// TwinCAT 3 PLC project M1L1_PLC
// ProgramVersion: 3.1.4020.5
// libraries:
//   Tc2_MC2, * (Beckhoff Automation GmbH)
//   Tc2_SerialCom, * (Beckhoff Automation GmbH)
//   Tc2_Standard, * (Beckhoff Automation GmbH)
//   Tc2_System, * (Beckhoff Automation GmbH)
//   Tc2_Utilities, * (Beckhoff Automation GmbH)
//   Tc3_Module, * (Beckhoff Automation GmbH)
//   VisuDialogs, * (System)
//   lcls-twincat-motion,0.0.0,SLAC
// project tree:
//   Common/POUs/Helpers/ FB_PI_E621_SerialDriver.TcPOU (not stored), FB_PI_E621_SerialTransaction.TcPOU (not stored)
//   DUTs/ DUT_MotionStage_Extras.TcDUT (not stored), ST_PiezoAxis.TcDUT (not stored)
//   / GlobalTextList.TcGTLO, PlcTask.TcTTO (not stored), serial_com.TcTTO, Visualization Manager.TcVMO (not stored)
//   GVLs/ GVL_SerialIO.TcGVL (not stored)
//   POUs/ MAIN.TcPOU
//   POUs/Serial Comm/ PiezoSerial.TcPOU, P_Serial_Com.TcPOU
//   VISUs/ Visualization.TcVIS, VISU_MotionStage.TcVIS (not stored)
// real-time tasks:
//   TASK PlcTask: cycle T#10ms, priority 20, ADS port 350
//   TASK serial_com: cycle T#10ms, priority 21, ADS port 351
// motion (NC):
//   TASK NC-Task 1 SAF: cycle T#2ms, priority 4, ADS port 501
//   TASK NC-Task 1 SVB: cycle T#10ms, priority 8, ADS port 511
//   AXIS y_up (id 6)
//     General: UnitName=um
//     Dynamic: Acceleration=5050, Deceleration=5050, Jerk=5100500, DelayTime=0.008
//     Velo: Maximum=100
//     OtherSettings: AllowMotionCmdToSlave=true
//     encoder EncType=29
//       EncPara: ScaleFactorNumerator=1, ScaleFactorDenominator=1000, MaxCount=#xffffffff, ReferenceSystem=1
//         SoftEndMinControl: Enable=true, Range=7200
//         SoftEndMaxControl: Enable=true, Range=100000
//         Inc: RefSoftSyncMask=#x0000ffff
//     drive DrvType=24
//       DrvPara: Inverse=true
//         Analog: VeloReferenz=500
//         TimeComp: TaskDelayCycles=1
//     controller CtrType=3
//       CtrPara: PriorControlFactor=1
//         PosDiffControl: Range=50, Time=0.2
//         PID: PosTn=0.005, PosIOutputLimit=0.0001, PosDOutputLimit=0, PosIDisableWhenMoving=true, DeadBandPosition=0.001
//         Observer: BandWidth=20
//   AXIS y_dwn (id 7)
//     General: UnitName=um
//     Dynamic: Acceleration=5050, Deceleration=5050, Jerk=5100500, DelayTime=0.008
//     Velo: Maximum=100
//     OtherSettings: AllowMotionCmdToSlave=true
//     encoder EncType=29
//       EncPara: ScaleFactorNumerator=1, ScaleFactorDenominator=1000, MaxCount=#xffffffff, ReferenceSystem=1
//         SoftEndMinControl: Enable=true, Range=10100
//         SoftEndMaxControl: Enable=true, Range=102600
//         Inc: RefSoftSyncMask=#x0000ffff
//     drive DrvType=24
//       DrvPara: Inverse=true
//         Analog: VeloReferenz=500
//         TimeComp: TaskDelayCycles=1
//     controller CtrType=3
//       CtrPara: PriorControlFactor=1
//         PosDiffControl: Range=50, Time=0.2
//         PID: PosTn=0.005, PosIOutputLimit=0.0001, PosDOutputLimit=0, PosIDisableWhenMoving=true, DeadBandPosition=0.001
//         Observer: BandWidth=20
//   AXIS x_up (id 1)
//     General: UnitName=um
//     Dynamic: Acceleration=1000, Deceleration=1000, DelayTime=0.008
//     Velo: Maximum=300
//     OtherSettings: AllowMotionCmdToSlave=true
//     encoder EncType=29
//       EncPara: ScaleFactorNumerator=0.001, MaxCount=#xffffffff, ReferenceSystem=1
//         SoftEndMinControl: Enable=true, Range=16900
//         SoftEndMaxControl: Enable=true, Range=23600
//         Inc: RefSoftSyncMask=#x0000ffff
//     drive DrvType=24
//       DrvPara: Inverse=true
//         Analog: VeloReferenz=625, ScaleFactorActTorque=0.1
//         TimeComp: TaskDelayCycles=1
//     controller CtrType=3
//       CtrPara: PriorControlFactor=1
//         PosDiffControl: Range=50
//         PID: PosTn=0.005, PosIOutputLimit=0.0001, PosDOutputLimit=0, PosIDisableWhenMoving=true, DeadBandPosition=0.001
//         Observer: BandWidth=20
//   AXIS x_dwn (id 9)
//     General: UnitName=um
//     Dynamic: AccelerationMaximum=1000, DecelerationMaximum=1000, Acceleration=1000, Deceleration=1000, Jerk=5000, DelayTime=0.008
//     Velo: Maximum=300
//     OtherSettings: AllowMotionCmdToSlave=true
//     encoder EncType=29
//       EncPara: ScaleFactorNumerator=0.001, MaxCount=#xffffffff
//         SoftEndMinControl: Enable=true, Range=15800
//         SoftEndMaxControl: Enable=true, Range=22600
//         Inc: RefSoftSyncMask=#x0000ffff
//     drive DrvType=24
//       Analog: VeloReferenz=625
//       TimeComp: TaskDelayCycles=1
//     controller CtrType=3
//       CtrPara: PriorControlFactor=1
//         PosDiffControl: Range=50, Time=0.2
//         PID: PosTn=0.005, PosIOutputLimit=0.0001, PosDOutputLimit=0, PosIDisableWhenMoving=true, DeadBandPosition=0.001
//         Observer: BandWidth=20
//   AXIS pitch (id 10)
//     General: UnitName=urad
//     Dynamic: Acceleration=64082.2, Deceleration=64082.2, Jerk=711156, DelayTime=0.008
//     Velo: Maximum=50
//     OtherSettings: AllowMotionCmdToSlave=true
//     encoder EncType=29
//       EncPara: ScaleFactorNumerator=0.00556, MaxCount=#xffffffff, ReferenceSystem=1
//         SoftEndMinControl: Enable=true, Range=57500
//         SoftEndMaxControl: Enable=true, Range=58900
//         ActPosCorrection: Time=0.008
//         Inc: RefSoftSyncMask=#x0000ffff
//     drive DrvType=24
//       DrvPara: Inverse=true
//         Analog: VeloReferenz=550
//         TimeComp: TaskDelayCycles=1
//     controller CtrType=3
//       CtrPara: PriorControlFactor=1
//         PosDiffControl: Range=15, Time=0.2
//         PID: PosKp=9, PosTn=0.0006, PosTv=1.2e-05, PosIOutputLimit=0.0005, PosDOutputLimit=0.0035, AccKa=0.001, DeadBandPosition=0.1
//         Observer: BandWidth=20
// I/O:
//   DEVICE Device 1 (EtherCAT)
//   DEVICE Device 4 (EtherCAT), AmsNetId 5.54.18.124.5.1
//     Term 4 (EK1100)
// variable links:
//   Axes/pitch <-> Device 4 (EtherCAT)/Term 4 (EK1100)/Term 10 (EL7047) - PitchCoarse
//     Drive/Inputs/In/nState1 @bit 3 <-> STM Status/Status/Error
//     Drive/Inputs/In/nState1 @bit 7 <-> STM Status/Status/Motor stall
//     Drive/Inputs/In/nState1 @bit 5 <-> STM Status/Status/Moving negative
//     Drive/Inputs/In/nState1 @bit 4 <-> STM Status/Status/Moving positive
//     Drive/Inputs/In/nState1 @bit 1 <-> STM Status/Status/Ready
//     Drive/Inputs/In/nState1 <-> STM Status/Status/Ready to enable
//     Drive/Inputs/In/nState1 @bit 6 <-> STM Status/Status/Torque reduced
//     Drive/Inputs/In/nState1 @bit 2 <-> STM Status/Status/Warning
//     Drive/Inputs/In/nState2 @bit 3 <-> STM Status/Status/Digital input 1
//     Drive/Inputs/In/nState2 @bit 4 <-> STM Status/Status/Digital input 2
//     Drive/Inputs/In/nState2 @bit 5 <-> STM Status/Status/Sync error
//     Drive/Inputs/In/nState2 @bit 7 <-> STM Status/Status/TxPDO Toggle
//     Drive/Inputs/In/nState4 @bit 1 <-> WcState/InputToggle
//     Drive/Inputs/In/nState4 <-> WcState/WcState
//     Drive/Outputs/Out/nCtrl1 <-> STM Control/Control/Enable
//     Drive/Outputs/Out/nCtrl1 @bit 2 <-> STM Control/Control/Reduce torque
//     Drive/Outputs/Out/nCtrl1 @bit 1 <-> STM Control/Control/Reset
//     Drive/Outputs/Out/nCtrl2 @bit 3 <-> STM Control/Control/Digital output 1
//     Drive/Outputs/Out/nDataOut2[0] <-> STM Velocity/Velocity
//   Axes/pitch <-> Device 4 (EtherCAT)/Term 4 (EK1100)/Term 13 (EL5042) - Pitch
//     Enc/Inputs/In/nComState @bit 1 <-> WcState/InputToggle
//     Enc/Inputs/In/nComState <-> WcState/WcState
//     Enc/Inputs/In/nDataIn1 <-> FB Inputs Channel 1/Position
//     Enc/Inputs/In/nState1 @bit 12 <-> FB Inputs Channel 1/Status/Diag
//     Enc/Inputs/In/nState1 @bit 1 <-> FB Inputs Channel 1/Status/Error
//     Enc/Inputs/In/nState1 @bit 14 <-> FB Inputs Channel 1/Status/Input cycle counter
//     Enc/Inputs/In/nState1 @bit 2 <-> FB Inputs Channel 1/Status/Ready
//     Enc/Inputs/In/nState1 @bit 13 <-> FB Inputs Channel 1/Status/TxPDO State
//     Enc/Inputs/In/nState1 <-> FB Inputs Channel 1/Status/Warning
//   Axes/x_dwn <-> Device 4 (EtherCAT)/Term 4 (EK1100)/Term 12 (EL5042) - X
//     Enc/Inputs/In/nComState @bit 1 <-> WcState/InputToggle
//     Enc/Inputs/In/nComState <-> WcState/WcState
//     Enc/Inputs/In/nDataIn1 <-> FB Inputs Channel 2/Position
//     Enc/Inputs/In/nState1 @bit 12 <-> FB Inputs Channel 2/Status/Diag
//     Enc/Inputs/In/nState1 @bit 1 <-> FB Inputs Channel 2/Status/Error
//     Enc/Inputs/In/nState1 @bit 14 <-> FB Inputs Channel 2/Status/Input cycle counter
//     Enc/Inputs/In/nState1 @bit 2 <-> FB Inputs Channel 2/Status/Ready
//     Enc/Inputs/In/nState1 @bit 13 <-> FB Inputs Channel 2/Status/TxPDO State
//     Enc/Inputs/In/nState1 <-> FB Inputs Channel 2/Status/Warning
//   Axes/x_dwn <-> Device 4 (EtherCAT)/Term 4 (EK1100)/Term 9 (EL7047) - Xdwn
//     Drive/Inputs/In/nState1 @bit 3 <-> STM Status/Status/Error
//     Drive/Inputs/In/nState1 @bit 7 <-> STM Status/Status/Motor stall
//     Drive/Inputs/In/nState1 @bit 5 <-> STM Status/Status/Moving negative
//     Drive/Inputs/In/nState1 @bit 4 <-> STM Status/Status/Moving positive
//     Drive/Inputs/In/nState1 @bit 1 <-> STM Status/Status/Ready
//     Drive/Inputs/In/nState1 <-> STM Status/Status/Ready to enable
//     Drive/Inputs/In/nState1 @bit 6 <-> STM Status/Status/Torque reduced
//     Drive/Inputs/In/nState1 @bit 2 <-> STM Status/Status/Warning
//     Drive/Inputs/In/nState2 @bit 3 <-> STM Status/Status/Digital input 1
//     Drive/Inputs/In/nState2 @bit 4 <-> STM Status/Status/Digital input 2
//     Drive/Inputs/In/nState2 @bit 5 <-> STM Status/Status/Sync error
//     Drive/Inputs/In/nState2 @bit 7 <-> STM Status/Status/TxPDO Toggle
//     Drive/Inputs/In/nState4 @bit 1 <-> WcState/InputToggle
//     Drive/Inputs/In/nState4 <-> WcState/WcState
//     Drive/Outputs/Out/nCtrl1 <-> STM Control/Control/Enable
//     Drive/Outputs/Out/nCtrl1 @bit 2 <-> STM Control/Control/Reduce torque
//     Drive/Outputs/Out/nCtrl1 @bit 1 <-> STM Control/Control/Reset
//     Drive/Outputs/Out/nCtrl2 @bit 3 <-> STM Control/Control/Digital output 1
//     Drive/Outputs/Out/nDataOut2[0] <-> STM Velocity/Velocity
//   Axes/y_dwn <-> Device 4 (EtherCAT)/Term 4 (EK1100)/Term 11 (EL5042) - Y
//     Enc/Inputs/In/nComState @bit 1 <-> WcState/InputToggle
//     Enc/Inputs/In/nComState <-> WcState/WcState
//     Enc/Inputs/In/nDataIn1 <-> FB Inputs Channel 2/Position
//     Enc/Inputs/In/nState1 @bit 12 <-> FB Inputs Channel 2/Status/Diag
//     Enc/Inputs/In/nState1 @bit 1 <-> FB Inputs Channel 2/Status/Error
//     Enc/Inputs/In/nState1 @bit 14 <-> FB Inputs Channel 2/Status/Input cycle counter
//     Enc/Inputs/In/nState1 @bit 2 <-> FB Inputs Channel 2/Status/Ready
//     Enc/Inputs/In/nState1 @bit 13 <-> FB Inputs Channel 2/Status/TxPDO State
//     Enc/Inputs/In/nState1 <-> FB Inputs Channel 2/Status/Warning
//   Axes/y_dwn <-> Device 4 (EtherCAT)/Term 4 (EK1100)/Term 7 (EL7047) - Ydwn
//     Drive/Inputs/In/nState1 @bit 3 <-> STM Status/Status/Error
//     Drive/Inputs/In/nState1 @bit 7 <-> STM Status/Status/Motor stall
//     Drive/Inputs/In/nState1 @bit 5 <-> STM Status/Status/Moving negative
//     Drive/Inputs/In/nState1 @bit 4 <-> STM Status/Status/Moving positive
//     Drive/Inputs/In/nState1 @bit 1 <-> STM Status/Status/Ready
//     Drive/Inputs/In/nState1 <-> STM Status/Status/Ready to enable
//     Drive/Inputs/In/nState1 @bit 6 <-> STM Status/Status/Torque reduced
//     Drive/Inputs/In/nState1 @bit 2 <-> STM Status/Status/Warning
//     Drive/Inputs/In/nState2 @bit 3 <-> STM Status/Status/Digital input 1
//     Drive/Inputs/In/nState2 @bit 4 <-> STM Status/Status/Digital input 2
//     Drive/Inputs/In/nState2 @bit 5 <-> STM Status/Status/Sync error
//     Drive/Inputs/In/nState2 @bit 7 <-> STM Status/Status/TxPDO Toggle
//     Drive/Inputs/In/nState4 @bit 1 <-> WcState/InputToggle
//     Drive/Inputs/In/nState4 <-> WcState/WcState
//     Drive/Outputs/Out/nCtrl1 <-> STM Control/Control/Enable
//     Drive/Outputs/Out/nCtrl1 @bit 2 <-> STM Control/Control/Reduce torque
//     Drive/Outputs/Out/nCtrl1 @bit 1 <-> STM Control/Control/Reset
//     Drive/Outputs/Out/nCtrl2 @bit 3 <-> STM Control/Control/Digital output 1
//     Drive/Outputs/Out/nDataOut2[0] <-> STM Velocity/Velocity
//   Axes/y_up <-> Device 4 (EtherCAT)/Term 4 (EK1100)/Term 11 (EL5042) - Y
//     Enc/Inputs/In/nComState @bit 1 <-> WcState/InputToggle
//     Enc/Inputs/In/nComState <-> WcState/WcState
//     Enc/Inputs/In/nDataIn1 <-> FB Inputs Channel 1/Position
//     Enc/Inputs/In/nState1 @bit 12 <-> FB Inputs Channel 1/Status/Diag
//     Enc/Inputs/In/nState1 @bit 1 <-> FB Inputs Channel 1/Status/Error
//     Enc/Inputs/In/nState1 @bit 14 <-> FB Inputs Channel 1/Status/Input cycle counter
//     Enc/Inputs/In/nState1 @bit 2 <-> FB Inputs Channel 1/Status/Ready
//     Enc/Inputs/In/nState1 @bit 13 <-> FB Inputs Channel 1/Status/TxPDO State
//     Enc/Inputs/In/nState1 <-> FB Inputs Channel 1/Status/Warning
//   Axes/y_up <-> Device 4 (EtherCAT)/Term 4 (EK1100)/Term 6 (EL7047) - Yup
//     Drive/Inputs/In/nState1 @bit 3 <-> STM Status/Status/Error
//     Drive/Inputs/In/nState1 @bit 7 <-> STM Status/Status/Motor stall
//     Drive/Inputs/In/nState1 @bit 5 <-> STM Status/Status/Moving negative
//     Drive/Inputs/In/nState1 @bit 4 <-> STM Status/Status/Moving positive
//     Drive/Inputs/In/nState1 @bit 1 <-> STM Status/Status/Ready
//     Drive/Inputs/In/nState1 <-> STM Status/Status/Ready to enable
//     Drive/Inputs/In/nState1 @bit 6 <-> STM Status/Status/Torque reduced
//     Drive/Inputs/In/nState1 @bit 2 <-> STM Status/Status/Warning
//     Drive/Inputs/In/nState2 @bit 3 <-> STM Status/Status/Digital input 1
//     Drive/Inputs/In/nState2 @bit 4 <-> STM Status/Status/Digital input 2
//     Drive/Inputs/In/nState2 @bit 5 <-> STM Status/Status/Sync error
//     Drive/Inputs/In/nState2 @bit 7 <-> STM Status/Status/TxPDO Toggle
//     Drive/Inputs/In/nState4 @bit 1 <-> WcState/InputToggle
//     Drive/Inputs/In/nState4 <-> WcState/WcState
//     Drive/Outputs/Out/nCtrl1 <-> STM Control/Control/Enable
//     Drive/Outputs/Out/nCtrl1 @bit 2 <-> STM Control/Control/Reduce torque
//     Drive/Outputs/Out/nCtrl1 @bit 1 <-> STM Control/Control/Reset
//     Drive/Outputs/Out/nCtrl2 @bit 3 <-> STM Control/Control/Digital output 1
//     Drive/Outputs/Out/nDataOut2[0] <-> STM Velocity/Velocity
//   (this object) <-> Device 4 (EtherCAT)/Term 4 (EK1100)/Term 12 (EL5042) - X
//     Enc/Inputs/In/nComState @bit 1 <-> WcState/InputToggle
//     Enc/Inputs/In/nComState <-> WcState/WcState
//     Enc/Inputs/In/nDataIn1 <-> FB Inputs Channel 1/Position
//     Enc/Inputs/In/nState1 @bit 12 <-> FB Inputs Channel 1/Status/Diag
//     Enc/Inputs/In/nState1 @bit 1 <-> FB Inputs Channel 1/Status/Error
//     Enc/Inputs/In/nState1 @bit 14 <-> FB Inputs Channel 1/Status/Input cycle counter
//     Enc/Inputs/In/nState1 @bit 2 <-> FB Inputs Channel 1/Status/Ready
//     Enc/Inputs/In/nState1 @bit 13 <-> FB Inputs Channel 1/Status/TxPDO State
//     Enc/Inputs/In/nState1 <-> FB Inputs Channel 1/Status/Warning
//   (this object) <-> Device 4 (EtherCAT)/Term 4 (EK1100)/Term 8 (EL7047) - Xup
//     Drive/Inputs/In/nState1 @bit 3 <-> STM Status/Error
//     Drive/Inputs/In/nState1 @bit 7 <-> STM Status/Motor stall
//     Drive/Inputs/In/nState1 @bit 5 <-> STM Status/Moving negative
//     Drive/Inputs/In/nState1 @bit 4 <-> STM Status/Moving positive
//     Drive/Inputs/In/nState1 @bit 1 <-> STM Status/Ready
//     Drive/Inputs/In/nState1 <-> STM Status/Ready to enable
//     Drive/Inputs/In/nState1 @bit 6 <-> STM Status/Torque reduced
//     Drive/Inputs/In/nState1 @bit 2 <-> STM Status/Warning
//     Drive/Inputs/In/nState2 @bit 3 <-> STM Status/Digital input 1
//     Drive/Inputs/In/nState2 @bit 4 <-> STM Status/Digital input 2
//     Drive/Inputs/In/nState2 @bit 5 <-> STM Status/Sync error
//     Drive/Inputs/In/nState2 @bit 7 <-> STM Status/TxPDO Toggle
//     Drive/Inputs/In/nState4 @bit 1 <-> WcState/InputToggle
//     Drive/Inputs/In/nState4 <-> WcState/WcState
//     Drive/Outputs/Out/nCtrl1 <-> STM Control/Enable
//     Drive/Outputs/Out/nCtrl1 @bit 2 <-> STM Control/Reduce torque
//     Drive/Outputs/Out/nCtrl1 @bit 1 <-> STM Control/Reset
//     Drive/Outputs/Out/nCtrl2 @bit 3 <-> STM Control/Digital output 1
//     Drive/Outputs/Out/nDataOut2[0] <-> STM Velocity/Velocity
//   M1L1_PLC Instance <-> Device 1 (EtherCAT)/Term 1 (EK1200)/Term 2 (EL1004)
//     PlcTask Inputs/MAIN.stoEnable1 <-> Channel 1/Input
//     PlcTask Inputs/MAIN.stoEnable2 <-> Channel 2/Input
//   M1L1_PLC Instance <-> Device 4 (EtherCAT)/Term 4 (EK1100)/Term 10 (EL7047) - PitchCoarse
//     PlcTask Inputs/MAIN.M5.bLimitBackwardEnable <-> STM Status/Status/Digital input 2
//     PlcTask Inputs/MAIN.M5.bLimitForwardEnable <-> STM Status/Status/Digital input 1
//   M1L1_PLC Instance <-> Device 4 (EtherCAT)/Term 4 (EK1100)/Term 11 (EL5042) - Y
//     PlcTask Inputs/MAIN.bEncWarningYdwn <-> FB Inputs Channel 2/Status/Warning
//     PlcTask Inputs/MAIN.bEncWarningYup <-> FB Inputs Channel 1/Status/Warning
//     PlcTask Inputs/MAIN.y_dwn_enc/Count <-> FB Inputs Channel 2/Position
//     PlcTask Inputs/MAIN.y_up_enc/Count <-> FB Inputs Channel 1/Position
//   M1L1_PLC Instance <-> Device 4 (EtherCAT)/Term 4 (EK1100)/Term 12 (EL5042) - X
//     PlcTask Inputs/MAIN.bEncWarningXdwn <-> FB Inputs Channel 2/Status/Warning
//     PlcTask Inputs/MAIN.x_dwn_enc/Count <-> FB Inputs Channel 2/Position
//     PlcTask Inputs/MAIN.x_up_enc/Count <-> FB Inputs Channel 1/Position
//   M1L1_PLC Instance <-> Device 4 (EtherCAT)/Term 4 (EK1100)/Term 13 (EL5042) - Pitch
//     PlcTask Inputs/MAIN.bEncWarningPitch <-> FB Inputs Channel 1/Status/Warning
//   M1L1_PLC Instance <-> Device 4 (EtherCAT)/Term 4 (EK1100)/Term 6 (EL7047) - Yup
//     PlcTask Inputs/MAIN.M1.bLimitBackwardEnable <-> STM Status/Status/Digital input 2
//     PlcTask Inputs/MAIN.M1.bLimitForwardEnable <-> STM Status/Status/Digital input 1
//   M1L1_PLC Instance <-> Device 4 (EtherCAT)/Term 4 (EK1100)/Term 7 (EL7047) - Ydwn
//     PlcTask Inputs/MAIN.M2.bLimitBackwardEnable <-> STM Status/Status/Digital input 2
//     PlcTask Inputs/MAIN.M2.bLimitForwardEnable <-> STM Status/Status/Digital input 1
//   M1L1_PLC Instance <-> Device 4 (EtherCAT)/Term 4 (EK1100)/Term 8 (EL7047) - Xup
//     PlcTask Inputs/MAIN.M3.bLimitBackwardEnable <-> STM Status/Digital input 2
//     PlcTask Inputs/MAIN.M3.bLimitForwardEnable <-> STM Status/Digital input 1
//   M1L1_PLC Instance <-> Device 4 (EtherCAT)/Term 4 (EK1100)/Term 9 (EL7047) - Xdwn
//     PlcTask Inputs/MAIN.M4.bLimitBackwardEnable <-> STM Status/Status/Digital input 2
//     PlcTask Inputs/MAIN.M4.bLimitForwardEnable <-> STM Status/Status/Digital input 1
//   M1L1_PLC Instance <-> NC-Task 1 SAF/Axes/pitch
//     PlcTask Inputs/MAIN.M5.Axis.NcToPlc <-> Outputs/ToPlc
//     PlcTask Outputs/MAIN.M5.Axis.PlcToNc <-> Inputs/FromPlc
//   M1L1_PLC Instance <-> NC-Task 1 SAF/Axes/x_dwn
//     PlcTask Inputs/MAIN.M4.Axis.NcToPlc <-> Outputs/ToPlc
//     PlcTask Outputs/MAIN.M4.Axis.PlcToNc <-> Inputs/FromPlc
//   M1L1_PLC Instance <-> NC-Task 1 SAF/Axes/x_up
//     PlcTask Inputs/MAIN.M3.Axis.NcToPlc <-> Outputs/ToPlc
//     PlcTask Outputs/MAIN.M3.Axis.PlcToNc <-> Inputs/FromPlc
//   M1L1_PLC Instance <-> NC-Task 1 SAF/Axes/y_dwn
//     PlcTask Inputs/MAIN.M2.Axis.NcToPlc <-> Outputs/ToPlc
//     PlcTask Outputs/MAIN.M2.Axis.PlcToNc <-> Inputs/FromPlc
//   M1L1_PLC Instance <-> NC-Task 1 SAF/Axes/y_up
//     PlcTask Inputs/MAIN.M1.Axis.NcToPlc <-> Outputs/ToPlc
//     PlcTask Outputs/MAIN.M1.Axis.PlcToNc <-> Inputs/FromPlc

CONFIGURATION M1L1_PLC
    RESOURCE PLC ON TwinCAT3
        TASK serial_com(INTERVAL := T#10ms, PRIORITY := 21);
        PROGRAM P_Serial_Com WITH serial_com : P_Serial_Com;
    END_RESOURCE
END_CONFIGURATION

// ---- POUs/Serial Comm/P_Serial_Com.TcPOU
PROGRAM P_Serial_Com
VAR
	fbSerialLineControl_EL6001_P1: SerialLineControl;
END_VAR

//These are the global IOs...don't forget to copy your data into them

(* EL6001 Serial port 0 com function *)
fbSerialLineControl_EL6001_P1(
	Mode:= SERIALLINEMODE_EL6_22B (*SERIALLINEMODE_KL6_22B_STANDARD*),
	pComIn:= ADR(Serial_P1_stComIn),
	pComOut:=ADR(Serial_P1_stComOut) ,
	SizeComIn:= SIZEOF(Serial_P1_stComIn),
	TxBuffer:= Serial_P1_SerialTXBuffer,
	RxBuffer:= Serial_P1_SerialRXBuffer,
	Error=> ,
	ErrorID=> );

END_PROGRAM

// ---- POUs/MAIN.TcPOU
PROGRAM MAIN
VAR
    M1: DUT_MotionStage:=(nCommand:=3); // Yup
	M2: DUT_MotionStage:=(nCommand:=3); // Ydwn
	M3: DUT_MotionStage:=(nCommand:=3); // Xup
	M4: DUT_MotionStage:=(nCommand:=3); // Xdwn
	M5: DUT_MotionStage:=(nCommand:=3); // PitchCoarse
	M1_Extras : DUT_MotionStage_Extras;
	M2_Extras : DUT_MotionStage_Extras;
	M3_Extras : DUT_MotionStage_Extras;
	M4_Extras : DUT_MotionStage_Extras;
	M5_Extras : DUT_MotionStage_Extras;

	fbMotionStage_x_up, fbMotionStage_x_dwn, fbMotionStage_y_up, fbMotionStage_y_dwn, fbMotionStage_pitch : FB_MotionStage;

	stoEnable1 AT %I* : BOOL;
	stoEnable2 AT %I* : BOOL;
	x_up_enc  AT %I*: ST_RenishawAbsEnc;
	x_dwn_enc  AT %I*: ST_RenishawAbsEnc;
	y_up_enc  AT %I*: ST_RenishawAbsEnc;
	y_dwn_enc  AT %I*: ST_RenishawAbsEnc;

	// Auto coupling function block
	fbAutoCoupleX : FB_GantryAutoCoupling;
	fbAutoCoupleY : FB_GantryAutoCoupling;
	bExecuteCoupleX : BOOL;
	bExecuteCoupleY : BOOL;
	bExecuteDecoupleX : BOOL;
	bExecuteDecoupleY : BOOL;
	bGantryAlreadyCoupledX : BOOL;
	bGantryAlreadyCoupledY : BOOL;
	
	// Gantry variables
	nCurrGantryX : LINT;
	nCurrGantryY : LINT;
	nGantryTolX : LINT := 75000;
	nGantryTolY : LINT := 75000;
	fCurrGantryX_um : LREAL;
	fCurrGantryY_um : LREAL;

	// Current Variables
	nCoilACurrRaw AT %I* : UINT;
	nCoilBCurrRaw AT %I* : UINT;
	nCoilACurr : INT;
	nCoilBCurr : INT;
	nTotCurr : INT;

	// Counters for encoder warning
	ctuXup : CTU;
	bEncWarningXup AT %I* : BOOL; // TRUE when encoder warning occurs
	nNumWarningsXup : WORD := 0;

	ctuXdwn : CTU;
	bEncWarningXdwn AT %I* : BOOL; // TRUE when encoder warning occurs
	nNumWarningsXdwn : WORD := 0;

	ctuYup : CTU;
	bEncWarningYup AT %I* : BOOL; // TRUE when encoder warning occurs
	nNumWarningsYup : WORD := 0;

	ctuYdwn : CTU;
	bEncWarningYdwn AT %I* : BOOL; // TRUE when encoder warning occurs
	nNumWarningsYdwn : WORD := 0;

	ctuPitch : CTU;
	bEncWarningPitch AT %I* : BOOL; // TRUE when encoder warning occurs
	nNumWarningsPitch : WORD := 0;
END_VAR

// M2K3
// Buttons to enable motors: write 0 to enable, 2 to disable
M1.nEnableMode; // Yup
M2.nEnableMode; // Ydwn
M3.nEnableMode; // Xup
M4.nEnableMode; // Xdwn
M5.nEnableMode; // PitchCoarse

// Encoder Reference Values: Initially took from Axilon FAT
// Had to realign encoders (lights were red) and so now using motor positions after aligning (lights turned blue)
// M2K3 Ref Vals
(*
y_up_enc.Ref := 43575680;
y_dwn_enc.Ref := 46974520;
x_up_enc.Ref := 20359920;
x_dwn_enc.Ref := 19780970;
*)
// Gantry zero positions after realignment with metrology
y_up_enc.Ref := 40653120;
y_dwn_enc.Ref := 43456180;
x_up_enc.Ref := 23635520;
x_dwn_enc.Ref := 22541650;

// Gantry Differences to monitor
nCurrGantryY := ((ULINT_TO_LINT(y_up_enc.Count) - ULINT_TO_LINT(y_up_enc.Ref)) - (ULINT_TO_LINT(y_dwn_enc.Count) - ULINT_TO_LINT(y_dwn_enc.Ref)));
nCurrGantryX := ((ULINT_TO_LINT(x_up_enc.Count) - ULINT_TO_LINT(x_up_enc.Ref)) - (ULINT_TO_LINT(x_dwn_enc.Count) - ULINT_TO_LINT(x_dwn_enc.Ref)));
fCurrGantryY_um := LINT_TO_LREAL(nCurrGantryY)/1000.0;
fCurrGantryx_um := LINT_TO_LREAL(nCurrGantryX)/1000.0;

// E-stop
M1.bHardwareEnable := stoEnable1 AND stoEnable2;
M2.bHardwareEnable := stoEnable1 AND stoEnable2;
M3.bHardwareEnable := stoEnable1 AND stoEnable2;
M4.bHardwareEnable := stoEnable1 AND stoEnable2;
M5.bHardwareEnable := stoEnable1 AND stoEnable2;


// Start Autocoupling
fbAutoCoupleX(nGantryTol:=nGantryTolX, Master:=M3, MasterEnc:=x_up_enc, Slave:=M4,
	          SlaveEnc:=x_dwn_enc, bExecuteCouple:=bExecuteCoupleX,
              bExecuteDecouple:=bExecuteDecoupleX,
              bGantryAlreadyCoupled=>bGantryAlreadyCoupledX);


fbAutoCoupleY(nGantryTol:=nGantryTolY, Master:=M1, MasterEnc:=y_up_enc, Slave:=M2,
	          SlaveEnc:=y_dwn_enc, bExecuteCouple:=bExecuteCoupleY,
              bExecuteDecouple:=bExecuteDecoupleY,
			  bGantryAlreadyCoupled=>bGantryAlreadyCoupledY);


fbMotionStage_y_up  (stMotionStage:=M1);
fbMotionStage_y_dwn (stMotionStage:=M2);
fbMotionStage_x_up  (stMotionStage:=M3);
fbMotionStage_x_dwn (stMotionStage:=M4);
fbMotionStage_pitch (stMotionStage:=M5);

// Record Coil Current
nCoilACurr := UINT_TO_INT(nCoilACurrRaw);
nCoilBCurr := UINT_TO_INT(nCoilBCurrRaw);
nTotCurr := ABS(nCoilACurr) + ABS(nCoilBCurr);

// Count when encoders throw warning
ctuXup(CU:=bEncWarningXup, CV=>nNumWarningsXup);
ctuXdwn(CU:=bEncWarningXdwn, CV=>nNumWarningsXdwn);
ctuYup(CU:=bEncWarningYup, CV=>nNumWarningsYup);
ctuYdwn(CU:=bEncWarningYdwn, CV=>nNumWarningsYdwn);
ctuPitch(CU:=bEncWarningPitch, CV=>nNumWarningsPitch);

END_PROGRAM

// ---- POUs/Serial Comm/PiezoSerial.TcPOU
PROGRAM PiezoSerial
VAR
	//PI Serial
	fbE621SerialDriverM1 : FB_PI_E621_SerialDriver;
	piezo: ST_PiezoAxis;
	rtInitParams	:	R_TRIG;
	tonTimeoutRstM1	: TON := (PT:=T#2S); //For timeout reset
	tonTimeoutRstM2	: TON := (PT:=T#2S); //For timeout reset
END_VAR

//M1 Piezo E-621
///////////////////////
	fbE621SerialDriverM1.i_xExecute := TRUE;
	fbE621SerialDriverM1.i_xExecute R= fbE621SerialDriverM1.q_xDone;
	fbE621SerialDriverM1(
		iq_stPiezoAxis:= piezo, 
		iq_stSerialRXBuffer:= Serial_P1_SerialRXBuffer, 
		iq_stSerialTXBuffer:= Serial_P1_SerialTXBuffer);

END_PROGRAM

// ---- GlobalTextList.TcGTLO
TEXTLIST GlobalTextList
  991 = '%f'
  359 = '%X'
  351 = '+'
  997 = '-'
  355 = '0 = Default Acceleration'
  357 = '0 = Default Deceleration'
  354 = 'Acceleration: %f'
  24 = 'Already Coupled: %f'
  349 = 'Clear'
  995 = 'Control'
  28 = 'Couple Motors'
  220 = 'Couple Status: 0 = Decoupled, 1 = Coupled'
  25 = 'Couple Status: TRUE if coupled'
  222 = 'Current Gantry Difference (Axilon): %f'
  27 = 'Current Gantry Difference in um'
  26 = 'Current Gantry Difference: %f'
  992 = 'Current Position'
  356 = 'Deceleration: %f'
  865 = 'Decouple Motors'
  217 = 'Disable'
  218 = 'Enable'
  863 = 'Enable Mode: %f'
  219 = 'Enable Status: 0 = Enabled, 2 = Disabled'
  221 = 'Ensure motors are coupled before attempting motion!'
  360 = 'Error Code'
  358 = 'Error:'
  999 = 'GO'
  348 = 'GO to set position'
  993 = 'High Limit Hit Indicator'
  990 = 'Low Limit Hit Indicator'
  994 = 'Moving:'
  860 = 'Pitch - MASTER'
  29 = 'Press To Couple Motors'
  866 = 'Press To Decouple Motors for independent control'
  996 = 'Set Position'
  352 = 'Settings'
  989 = 'Status'
  998 = 'Step Size'
  350 = 'STOP'
  861 = 'Units: um'
  862 = 'Units: urad'
  353 = 'Velocity: %f'
  864 = 'Write 0 to Enable, 2 to Disable'
  859 = 'Xdwn - SLAVE'
  858 = 'Xup - MASTER'
  771 = 'Ydwn - SLAVE'
  22 = 'Yleft - MASTER'
  23 = 'Yright - SLAVE'
  488 = 'Yup - MASTER'
END_TEXTLIST

// ---- VISUs/Visualization.TcVIS
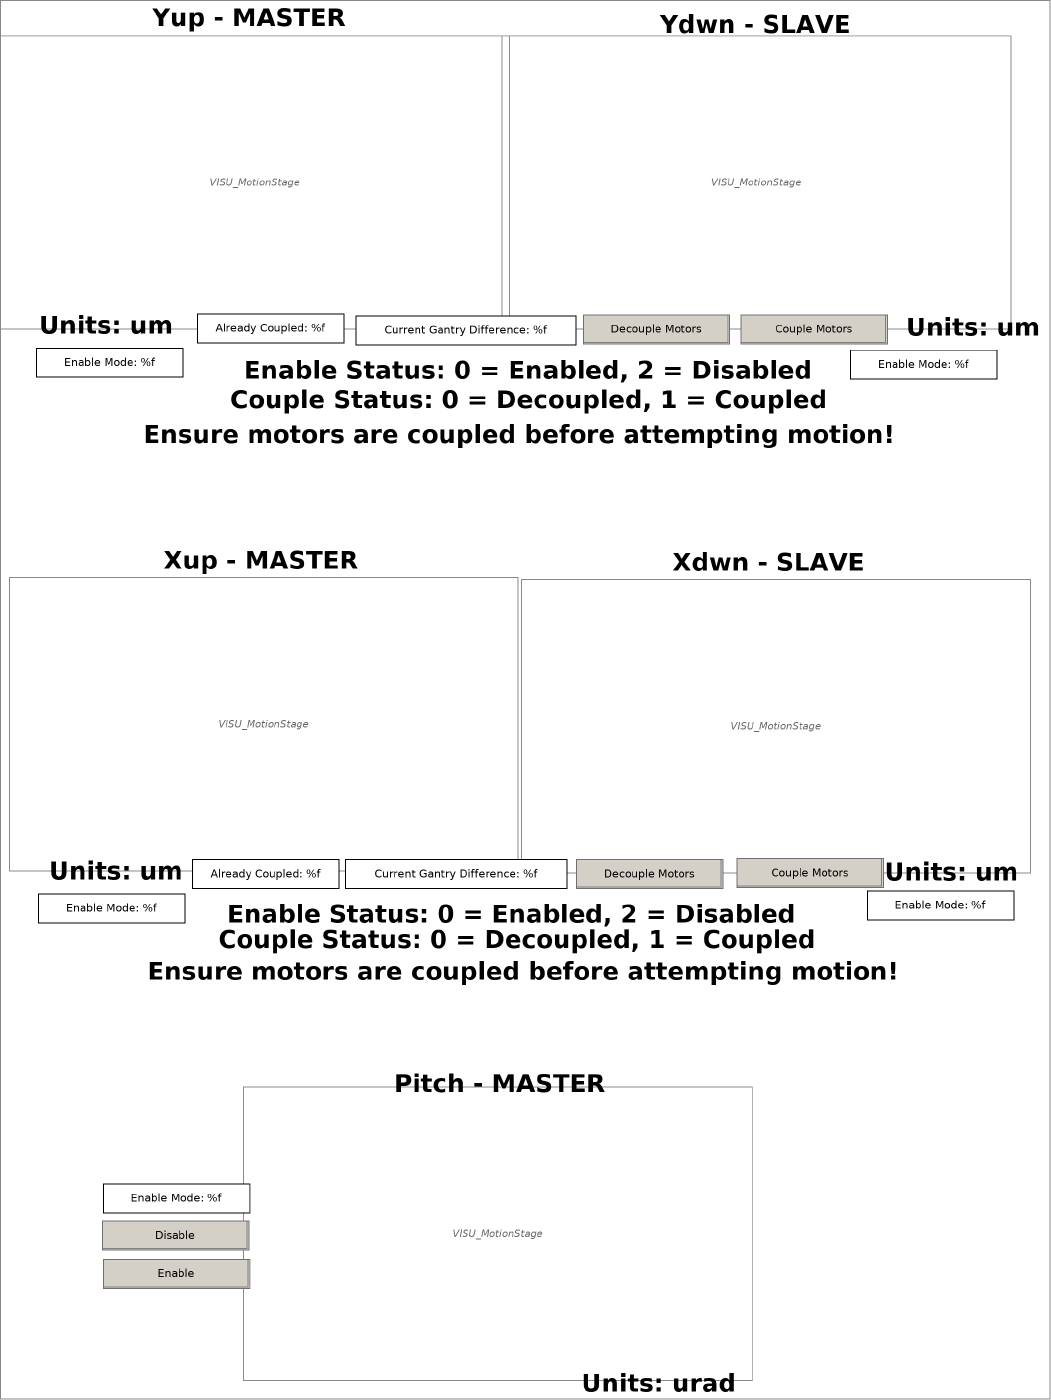
VISUALIZATION Visualization  // 1073x1429
    Label (14,2 481x31), "Yup - MASTER"
    Frame (0,36 520x300)
        shows VISU_MotionStage(VisuMotionStage := MAIN.M1, Extras := MAIN.M1_Extras)
    Frame (512,36 520x300)
        shows VISU_MotionStage(VisuMotionStage := MAIN.M2, Extras := MAIN.M2_Extras)
    Label (531,9 481x31), "Ydwn - SLAVE"
    Rectangle (201,320 150x30), "Already Coupled: %f", tooltip "Couple Status: TRUE if coupled", text variable: MAIN.bGantryAlreadyCoupledY
    Rectangle (363,322 225x30), "Current Gantry Difference: %f", tooltip "Current Gantry Difference in um", text variable: MAIN.fCurrGantryY_um
    Button (756,321 150x30), "Couple Motors", tooltip "Press To Couple Motors", text variable: MAIN.bExecuteCoupleY
        OnMouseDown: execute { MAIN.bExecuteCoupleY := TRUE; }
    Frame (9,589 520x300)
        shows VISU_MotionStage(VisuMotionStage := MAIN.M3, Extras := MAIN.M3_Extras)
    Label (26,556 481x31), "Xup - MASTER"
    Frame (532,591 520x300)
        shows VISU_MotionStage(VisuMotionStage := MAIN.M4, Extras := MAIN.M4_Extras)
    Label (544,558 481x31), "Xdwn - SLAVE"
    Rectangle (196,877 150x30), "Already Coupled: %f", tooltip "Couple Status: TRUE if coupled", text variable: MAIN.bGantryAlreadyCoupledX
    Rectangle (352,877 227x30), "Current Gantry Difference: %f", tooltip "Current Gantry Difference in um", text variable: MAIN.fCurrGantryX_um
    Frame (248,1109 520x300)
        shows VISU_MotionStage(VisuMotionStage := MAIN.M5, Extras := MAIN.M5_Extras)
    Label (270,1090 481x31), "Pitch - MASTER"
    Label (31,316 155x31), "Units: um"
    Label (916,318 155x31), "Units: um"
    Label (41,873 155x31), "Units: um"
    Label (894,874 155x31), "Units: um"
    Label (595,1396 155x31), "Units: urad"
    Rectangle (37,355 150x30), "Enable Mode: %f", tooltip "Write 0 to Enable, 2 to Disable", text variable: MAIN.M1.nEnableMode
    Rectangle (868,357 150x30), "Enable Mode: %f", tooltip "Write 0 to Enable, 2 to Disable", text variable: MAIN.M2.nEnableMode
    Button (595,321 150x30), "Decouple Motors", tooltip "Press To Decouple Motors for independent control"
        OnMouseDown: execute { MAIN.bExecuteDecoupleY := TRUE; }
    Button (588,877 150x30), "Decouple Motors", tooltip "Press To Decouple Motors for independent control"
        OnMouseDown: execute { MAIN.bExecuteDecoupleX := TRUE; }
    Button (752,876 150x30), "Couple Motors", tooltip "Press To Couple Motors", text variable: MAIN.bExecuteCoupleY
        OnMouseDown: execute { MAIN.bExecuteCoupleX := TRUE; }
    Rectangle (39,912 150x30), "Enable Mode: %f", tooltip "Write 0 to Enable, 2 to Disable", text variable: MAIN.M3.nEnableMode
    Rectangle (885,909 150x30), "Enable Mode: %f", tooltip "Write 0 to Enable, 2 to Disable", text variable: MAIN.M4.nEnableMode
    Rectangle (105,1208 150x30), "Enable Mode: %f", tooltip "Write 0 to Enable, 2 to Disable", text variable: MAIN.M5.nEnableMode
    Button (104,1246 150x30), "Disable"
        OnMouseDown: execute { MAIN.M5.nEnableMode := 2; }
    Button (105,1285 150x30), "Enable", colour toggle: MAIN.bExecuteDecoupleY
        OnMouseDown: execute { MAIN.M5.nEnableMode := 0; }
    Label (255,362 568x31), "Enable Status: 0 = Enabled, 2 = Disabled"
    Label (247,392 586x31), "Couple Status: 0 = Decoupled, 1 = Coupled"
    Label (238,917 568x31), "Enable Status: 0 = Enabled, 2 = Disabled"
    Label (235,943 586x31), "Couple Status: 0 = Decoupled, 1 = Coupled"
    Label (150,428 760x30), "Ensure motors are coupled before attempting motion!"
    Label (154,976 760x30), "Ensure motors are coupled before attempting motion!"
END_VISUALIZATION
